{attribute 'GeneratedUsingTerminal: EL3783-0000-0018'}
{attribute addProperty BoxType "EL3783-0000-0018"}
{attribute addProperty Id "L1_Voltage_StatusAT %I*L1_Voltage_Status_7371B0437L1_Voltage_SamplesAT %I*L1_Voltage_Samples_A8076B5D40L1_Current_StatusAT %I*L1_Current_Status_82DECBF67L1_Current_SamplesAT %I*L1_Current_Samples_7769579C40L2_Voltage_StatusAT %I*L2_Voltage_Status_0D1813FE7L2_Voltage_SamplesAT %I*L2_Voltage_Samples_9C71EF0D40L2_Current_StatusAT %I*L2_Current_Status_FCB7684B7L2_Current_SamplesAT %I*L2_Current_Samples_431FD3CC40L3_Voltage_StatusAT %I*L3_Voltage_Status_273F72957L3_Voltage_SamplesAT %I*L3_Voltage_Samples_8FA3933D40L3_Current_StatusAT %I*L3_Current_Status_D69009207L3_Current_SamplesAT %I*L3_Current_Samples_50CDAFFC40AI_NextSync1TimeAT %I*AI_NextSync1Time_6DC4D2968AI_Sample_CountAT %I*AI_Sample_Count_EA88CAD92AI_Current_RangeAT %I*AI_Current_Range_9DEBDE6D5WcStateAT %I*WcState_9091E0EB2InfoDataAT %I*InfoData_BEF6B88E18"}
{attribute addProperty CRC "1412900171"}
{attribute addProperty Size "317"}
TYPE EL3783_5437254B EXTENDS EtcSlaveTerminalBase_947E5A46 :
STRUCT
	{attribute addProperty Name "L1_Voltage_Status"}
	L1_Voltage_Status : L1_Voltage_Status_7371B043;
	{attribute addProperty Name "L1_Voltage_Samples"}
	L1_Voltage_Samples : L1_Voltage_Samples_A8076B5D;
	{attribute addProperty Name "L1_Current_Status"}
	L1_Current_Status : L1_Current_Status_82DECBF6;
	{attribute addProperty Name "L1_Current_Samples"}
	L1_Current_Samples : L1_Current_Samples_7769579C;
	{attribute addProperty Name "L2_Voltage_Status"}
	L2_Voltage_Status : L2_Voltage_Status_0D1813FE;
	{attribute addProperty Name "L2_Voltage_Samples"}
	L2_Voltage_Samples : L2_Voltage_Samples_9C71EF0D;
	{attribute addProperty Name "L2_Current_Status"}
	L2_Current_Status : L2_Current_Status_FCB7684B;
	{attribute addProperty Name "L2_Current_Samples"}
	L2_Current_Samples : L2_Current_Samples_431FD3CC;
	{attribute addProperty Name "L3_Voltage_Status"}
	L3_Voltage_Status : L3_Voltage_Status_273F7295;
	{attribute addProperty Name "L3_Voltage_Samples"}
	L3_Voltage_Samples : L3_Voltage_Samples_8FA3933D;
	{attribute addProperty Name "L3_Current_Status"}
	L3_Current_Status : L3_Current_Status_D6900920;
	{attribute addProperty Name "L3_Current_Samples"}
	L3_Current_Samples : L3_Current_Samples_50CDAFFC;
	{attribute addProperty Name "AI_NextSync1Time"}
	AI_NextSync1Time : AI_NextSync1Time_6DC4D296;
	{attribute addProperty Name "AI_Sample_Count"}
	AI_Sample_Count : AI_Sample_Count_EA88CAD9;
	{attribute addProperty Name "AI_Current_Range"}
	AI_Current_Range : AI_Current_Range_9DEBDE6D;
	{attribute addProperty Name "WcState"}
	WcState : WcState_9091E0EB;
	{attribute addProperty Name "InfoData"}
	InfoData : InfoData_BEF6B88E;
END_STRUCT
END_TYPE

(* stored: Version 1.2.0.0, ProductVersion 3.1.4024.9
   DUT EL3783_5437254B: Id {59cfdfe9-3c69-4b7e-a9f0-0f4da4d02f44} *)
